// TIA Portal project "Lamp e pulsanti" (V18)

(* hardware
DEVICE "S71500/ET200MP station_1"  S7-1500 station
   slot 0: "Telaio di montaggio_0"  Rack  6ES7 590-1***0-0AA0
   slot 1: "PLC_1"  CPU 1516-3 PN/DP  6ES7 516-3AN01-0AB0  V1.8
      slot 3: "Display CPU_1"  6ES7591-1BA00-0AA0
   slot 2: "DI 32x24VDC HF_1"  DI 32x24VDC HF  6ES7 521-1BL00-0AB0  V1.0
   slot 3: "DQ 32x24VDC/0.5A HF_1"  DQ 32x24VDC/0.5A HF  6ES7 522-1BL01-0AB0  V1.0
   slot 4: "AI 8xU/I/RTD/TC ST_1"  AI 8xU/I/RTD/TC ST  6ES7 531-7KF00-0AB0  V1.0
   slot 5: "AQ 4xU/I ST_1"  AQ 4xU/I ST  6ES7 532-5HD00-0AB0  V1.0
*)

// ===== PLC "PLC_1"  CPU 1516-3 PN/DP =====

VAR_GLOBAL   // PLC tag table "Tabella delle variabili standard"
   "P1" AT %M0.0 : Bool;   // Pulsante virtuale 1
   "P2" AT %M0.1 : Bool;   // Pulsante virtuale 2
   "LAMP1" AT %Q0.0 : Bool;   // Lampada/Led 1
   "LAMP2" AT %Q0.1 : Bool;   // Lampada/Led 2
   "LAMP3" AT %Q0.2 : Bool;   // Lampada/Led 3
   "LAMP4" AT %Q0.3 : Bool;   // Lampada/Led 4
END_VAR

ORGANIZATION_BLOCK "Main"   // OB1, LAD, ProgramCycle
TITLE = "Main Program Sweep (Cycle)"
{ S7_Optimized_Access := 'TRUE' }
VERSION : 0.1
   VAR_INPUT
      Initial_Call : Bool;   // Initial call of this OB
      Remanence : Bool;   // =True, if remanent data are available
   END_VAR
BEGIN

REGION Network 1: Lampada/Led 1
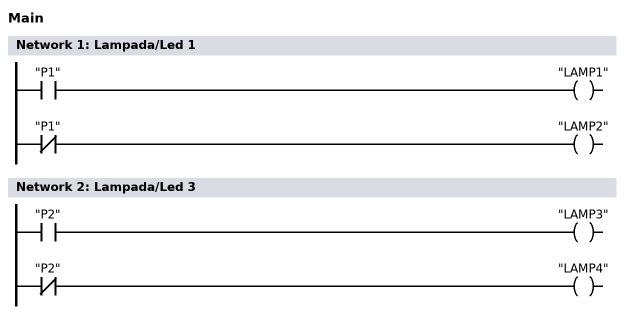
   RUNG wire#powerrail
      Contact( "P1" )
      Coil( "LAMP1" )
   END_RUNG
   RUNG wire#powerrail
      I_Contact( "P1" )
      Coil( "LAMP2" )
   END_RUNG
   // the same network as SCL:
   "LAMP1" := "P1";
   "LAMP2" := NOT "P1";
END_REGION

REGION Network 2: Lampada/Led 3
   RUNG wire#powerrail
      Contact( "P2" )
      Coil( "LAMP3" )
   END_RUNG
   RUNG wire#powerrail
      I_Contact( "P2" )
      Coil( "LAMP4" )
   END_RUNG
   // the same network as SCL:
   "LAMP3" := "P2";
   "LAMP4" := NOT "P2";
END_REGION
END_ORGANIZATION_BLOCK